{attribute 'pack_mode' := '1'}
TYPE ST_Result :
	STRUCT
		Busy	: BOOL;
		Error	: BOOL;
		Done	: BOOL;
		ErrorId : DINT;
	END_STRUCT
END_TYPE

(* stored: Version 1.1.0.1, ProductVersion 3.1.4024.12
   DUT ST_Result: Id {59ca350b-e84b-4e7f-9994-4868acbee99d} *)
